// TIA Portal V19 export
FUNCTION "MFG OUTPUT SECTION" : Void   // FC10, LAD
{ S7_Optimized_Access := 'TRUE' }
// stored: SetENOAutomatically false
   VAR_TEMP   // added for the SCL form of the ladder/FBD networks
      _w1 : Bool;
   END_VAR
BEGIN

REGION Network 1: PSFV-1 – OPEN
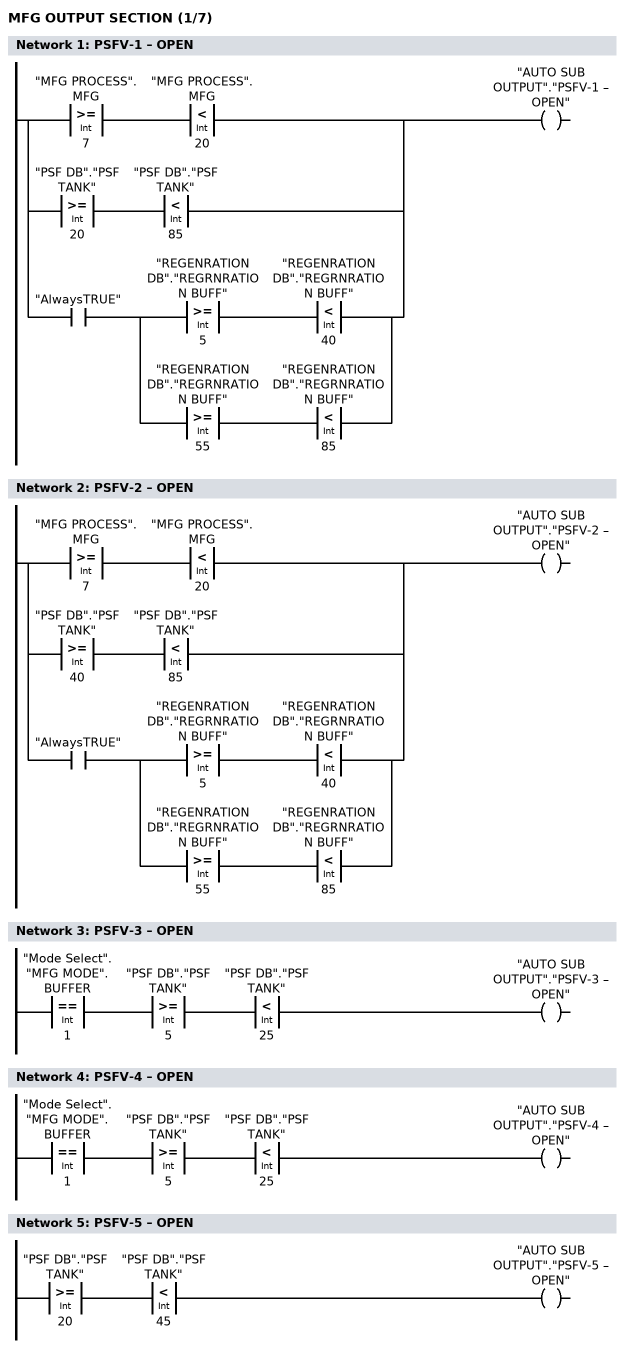
   RUNG wire#powerrail
      { S7_Templates := "SrcType := Int" } GE_Contact(in1 := "MFG PROCESS".MFG, in2 := 7)
      { S7_Templates := "SrcType := Int" } LT_Contact(in1 := "MFG PROCESS".MFG, in2 := 20)
      wire#w1
      Coil( "AUTO SUB OUTPUT"."PSFV-1 – OPEN" )
   END_RUNG
   RUNG wire#powerrail
      { S7_Templates := "SrcType := Int" } GE_Contact(in1 := "PSF DB"."PSF TANK", in2 := 20)
      { S7_Templates := "SrcType := Int" } LT_Contact(in1 := "PSF DB"."PSF TANK", in2 := 85)
   END_RUNG wire#w1
   RUNG wire#powerrail
      Contact( "AlwaysTRUE" )
      wire#w2
      { S7_Templates := "SrcType := Int" } GE_Contact(in1 := "REGENRATION DB"."REGRNRATION BUFF", in2 := 5)
      { S7_Templates := "SrcType := Int" } LT_Contact(in1 := "REGENRATION DB"."REGRNRATION BUFF", in2 := 40)
   END_RUNG wire#w1
   RUNG wire#w2
      { S7_Templates := "SrcType := Int" } GE_Contact(in1 := "REGENRATION DB"."REGRNRATION BUFF", in2 := 55)
      { S7_Templates := "SrcType := Int" } LT_Contact(in1 := "REGENRATION DB"."REGRNRATION BUFF", in2 := 85)
   END_RUNG wire#w1
   // the same network as SCL:
   "AUTO SUB OUTPUT"."PSFV-1 – OPEN" := (("MFG PROCESS".MFG >= 7) AND ("MFG PROCESS".MFG < 20)) OR (("PSF DB"."PSF TANK" >= 20) AND ("PSF DB"."PSF TANK" < 85)) OR ("AlwaysTRUE" AND ((("REGENRATION DB"."REGRNRATION BUFF" >= 5) AND ("REGENRATION DB"."REGRNRATION BUFF" < 40)) OR (("REGENRATION DB"."REGRNRATION BUFF" >= 55) AND ("REGENRATION DB"."REGRNRATION BUFF" < 85))));
END_REGION

REGION Network 2: PSFV-2 – OPEN
   RUNG wire#powerrail
      { S7_Templates := "SrcType := Int" } GE_Contact(in1 := "MFG PROCESS".MFG, in2 := 7)
      { S7_Templates := "SrcType := Int" } LT_Contact(in1 := "MFG PROCESS".MFG, in2 := 20)
      wire#w1
      Coil( "AUTO SUB OUTPUT"."PSFV-2 – OPEN" )
   END_RUNG
   RUNG wire#powerrail
      { S7_Templates := "SrcType := Int" } GE_Contact(in1 := "PSF DB"."PSF TANK", in2 := 40)
      { S7_Templates := "SrcType := Int" } LT_Contact(in1 := "PSF DB"."PSF TANK", in2 := 85)
   END_RUNG wire#w1
   RUNG wire#powerrail
      Contact( "AlwaysTRUE" )
      wire#w2
      { S7_Templates := "SrcType := Int" } GE_Contact(in1 := "REGENRATION DB"."REGRNRATION BUFF", in2 := 5)
      { S7_Templates := "SrcType := Int" } LT_Contact(in1 := "REGENRATION DB"."REGRNRATION BUFF", in2 := 40)
   END_RUNG wire#w1
   RUNG wire#w2
      { S7_Templates := "SrcType := Int" } GE_Contact(in1 := "REGENRATION DB"."REGRNRATION BUFF", in2 := 55)
      { S7_Templates := "SrcType := Int" } LT_Contact(in1 := "REGENRATION DB"."REGRNRATION BUFF", in2 := 85)
   END_RUNG wire#w1
   // the same network as SCL:
   "AUTO SUB OUTPUT"."PSFV-2 – OPEN" := (("MFG PROCESS".MFG >= 7) AND ("MFG PROCESS".MFG < 20)) OR (("PSF DB"."PSF TANK" >= 40) AND ("PSF DB"."PSF TANK" < 85)) OR ("AlwaysTRUE" AND ((("REGENRATION DB"."REGRNRATION BUFF" >= 5) AND ("REGENRATION DB"."REGRNRATION BUFF" < 40)) OR (("REGENRATION DB"."REGRNRATION BUFF" >= 55) AND ("REGENRATION DB"."REGRNRATION BUFF" < 85))));
END_REGION

REGION Network 3: PSFV-3 – OPEN
   RUNG wire#powerrail
      { S7_Templates := "SrcType := Int" } EQ_Contact(in1 := "Mode Select"."MFG MODE".BUFFER, in2 := 1)
      { S7_Templates := "SrcType := Int" } GE_Contact(in1 := "PSF DB"."PSF TANK", in2 := 5)
      { S7_Templates := "SrcType := Int" } LT_Contact(in1 := "PSF DB"."PSF TANK", in2 := 25)
      Coil( "AUTO SUB OUTPUT"."PSFV-3 – OPEN" )
   END_RUNG
   // the same network as SCL:
   "AUTO SUB OUTPUT"."PSFV-3 – OPEN" := ("Mode Select"."MFG MODE".BUFFER = 1) AND ("PSF DB"."PSF TANK" >= 5) AND ("PSF DB"."PSF TANK" < 25);
END_REGION

REGION Network 4: PSFV-4 – OPEN
   RUNG wire#powerrail
      { S7_Templates := "SrcType := Int" } EQ_Contact(in1 := "Mode Select"."MFG MODE".BUFFER, in2 := 1)
      { S7_Templates := "SrcType := Int" } GE_Contact(in1 := "PSF DB"."PSF TANK", in2 := 5)
      { S7_Templates := "SrcType := Int" } LT_Contact(in1 := "PSF DB"."PSF TANK", in2 := 25)
      Coil( "AUTO SUB OUTPUT"."PSFV-4 – OPEN" )
   END_RUNG
   // the same network as SCL:
   "AUTO SUB OUTPUT"."PSFV-4 – OPEN" := ("Mode Select"."MFG MODE".BUFFER = 1) AND ("PSF DB"."PSF TANK" >= 5) AND ("PSF DB"."PSF TANK" < 25);
END_REGION

REGION Network 5: PSFV-5 – OPEN
   RUNG wire#powerrail
      { S7_Templates := "SrcType := Int" } GE_Contact(in1 := "PSF DB"."PSF TANK", in2 := 20)
      { S7_Templates := "SrcType := Int" } LT_Contact(in1 := "PSF DB"."PSF TANK", in2 := 45)
      Coil( "AUTO SUB OUTPUT"."PSFV-5 – OPEN" )
   END_RUNG
   // the same network as SCL:
   "AUTO SUB OUTPUT"."PSFV-5 – OPEN" := ("PSF DB"."PSF TANK" >= 20) AND ("PSF DB"."PSF TANK" < 45);
END_REGION

REGION Network 6: PSFV-6 – OPEN
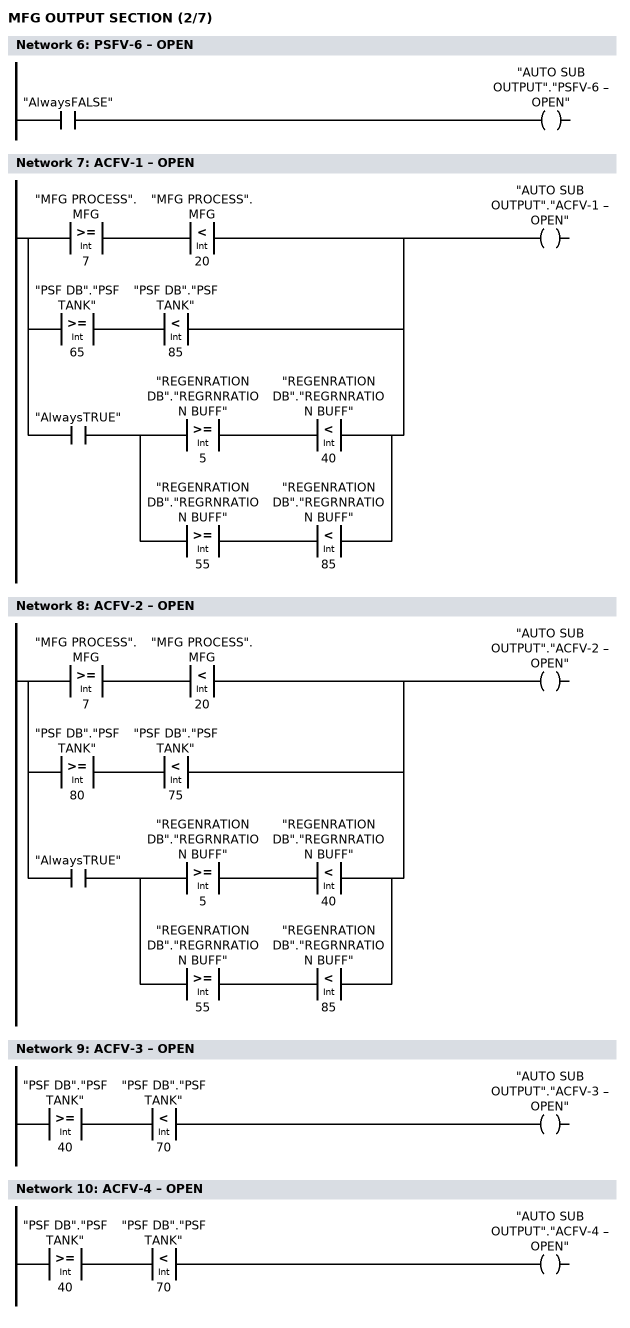
   RUNG wire#powerrail
      Contact( "AlwaysFALSE" )
      Coil( "AUTO SUB OUTPUT"."PSFV-6 – OPEN" )
   END_RUNG
   // the same network as SCL:
   "AUTO SUB OUTPUT"."PSFV-6 – OPEN" := "AlwaysFALSE";
END_REGION

REGION Network 7: ACFV-1 – OPEN
   RUNG wire#powerrail
      { S7_Templates := "SrcType := Int" } GE_Contact(in1 := "MFG PROCESS".MFG, in2 := 7)
      { S7_Templates := "SrcType := Int" } LT_Contact(in1 := "MFG PROCESS".MFG, in2 := 20)
      wire#w1
      Coil( "AUTO SUB OUTPUT"."ACFV-1 – OPEN" )
   END_RUNG
   RUNG wire#powerrail
      { S7_Templates := "SrcType := Int" } GE_Contact(in1 := "PSF DB"."PSF TANK", in2 := 65)
      { S7_Templates := "SrcType := Int" } LT_Contact(in1 := "PSF DB"."PSF TANK", in2 := 85)
   END_RUNG wire#w1
   RUNG wire#powerrail
      Contact( "AlwaysTRUE" )
      wire#w2
      { S7_Templates := "SrcType := Int" } GE_Contact(in1 := "REGENRATION DB"."REGRNRATION BUFF", in2 := 5)
      { S7_Templates := "SrcType := Int" } LT_Contact(in1 := "REGENRATION DB"."REGRNRATION BUFF", in2 := 40)
   END_RUNG wire#w1
   RUNG wire#w2
      { S7_Templates := "SrcType := Int" } GE_Contact(in1 := "REGENRATION DB"."REGRNRATION BUFF", in2 := 55)
      { S7_Templates := "SrcType := Int" } LT_Contact(in1 := "REGENRATION DB"."REGRNRATION BUFF", in2 := 85)
   END_RUNG wire#w1
   // the same network as SCL:
   "AUTO SUB OUTPUT"."ACFV-1 – OPEN" := (("MFG PROCESS".MFG >= 7) AND ("MFG PROCESS".MFG < 20)) OR (("PSF DB"."PSF TANK" >= 65) AND ("PSF DB"."PSF TANK" < 85)) OR ("AlwaysTRUE" AND ((("REGENRATION DB"."REGRNRATION BUFF" >= 5) AND ("REGENRATION DB"."REGRNRATION BUFF" < 40)) OR (("REGENRATION DB"."REGRNRATION BUFF" >= 55) AND ("REGENRATION DB"."REGRNRATION BUFF" < 85))));
END_REGION

REGION Network 8: ACFV-2 – OPEN
   RUNG wire#powerrail
      { S7_Templates := "SrcType := Int" } GE_Contact(in1 := "MFG PROCESS".MFG, in2 := 7)
      { S7_Templates := "SrcType := Int" } LT_Contact(in1 := "MFG PROCESS".MFG, in2 := 20)
      wire#w1
      Coil( "AUTO SUB OUTPUT"."ACFV-2 – OPEN" )
   END_RUNG
   RUNG wire#powerrail
      { S7_Templates := "SrcType := Int" } GE_Contact(in1 := "PSF DB"."PSF TANK", in2 := 80)
      { S7_Templates := "SrcType := Int" } LT_Contact(in1 := "PSF DB"."PSF TANK", in2 := 75)
   END_RUNG wire#w1
   RUNG wire#powerrail
      Contact( "AlwaysTRUE" )
      wire#w2
      { S7_Templates := "SrcType := Int" } GE_Contact(in1 := "REGENRATION DB"."REGRNRATION BUFF", in2 := 5)
      { S7_Templates := "SrcType := Int" } LT_Contact(in1 := "REGENRATION DB"."REGRNRATION BUFF", in2 := 40)
   END_RUNG wire#w1
   RUNG wire#w2
      { S7_Templates := "SrcType := Int" } GE_Contact(in1 := "REGENRATION DB"."REGRNRATION BUFF", in2 := 55)
      { S7_Templates := "SrcType := Int" } LT_Contact(in1 := "REGENRATION DB"."REGRNRATION BUFF", in2 := 85)
   END_RUNG wire#w1
   // the same network as SCL:
   "AUTO SUB OUTPUT"."ACFV-2 – OPEN" := (("MFG PROCESS".MFG >= 7) AND ("MFG PROCESS".MFG < 20)) OR (("PSF DB"."PSF TANK" >= 80) AND ("PSF DB"."PSF TANK" < 75)) OR ("AlwaysTRUE" AND ((("REGENRATION DB"."REGRNRATION BUFF" >= 5) AND ("REGENRATION DB"."REGRNRATION BUFF" < 40)) OR (("REGENRATION DB"."REGRNRATION BUFF" >= 55) AND ("REGENRATION DB"."REGRNRATION BUFF" < 85))));
END_REGION

REGION Network 9: ACFV-3 – OPEN
   RUNG wire#powerrail
      { S7_Templates := "SrcType := Int" } GE_Contact(in1 := "PSF DB"."PSF TANK", in2 := 40)
      { S7_Templates := "SrcType := Int" } LT_Contact(in1 := "PSF DB"."PSF TANK", in2 := 70)
      Coil( "AUTO SUB OUTPUT"."ACFV-3 – OPEN" )
   END_RUNG
   // the same network as SCL:
   "AUTO SUB OUTPUT"."ACFV-3 – OPEN" := ("PSF DB"."PSF TANK" >= 40) AND ("PSF DB"."PSF TANK" < 70);
END_REGION

REGION Network 10: ACFV-4 – OPEN
   RUNG wire#powerrail
      { S7_Templates := "SrcType := Int" } GE_Contact(in1 := "PSF DB"."PSF TANK", in2 := 40)
      { S7_Templates := "SrcType := Int" } LT_Contact(in1 := "PSF DB"."PSF TANK", in2 := 70)
      Coil( "AUTO SUB OUTPUT"."ACFV-4 – OPEN" )
   END_RUNG
   // the same network as SCL:
   "AUTO SUB OUTPUT"."ACFV-4 – OPEN" := ("PSF DB"."PSF TANK" >= 40) AND ("PSF DB"."PSF TANK" < 70);
END_REGION

REGION Network 11: ACFV-5 – OPEN
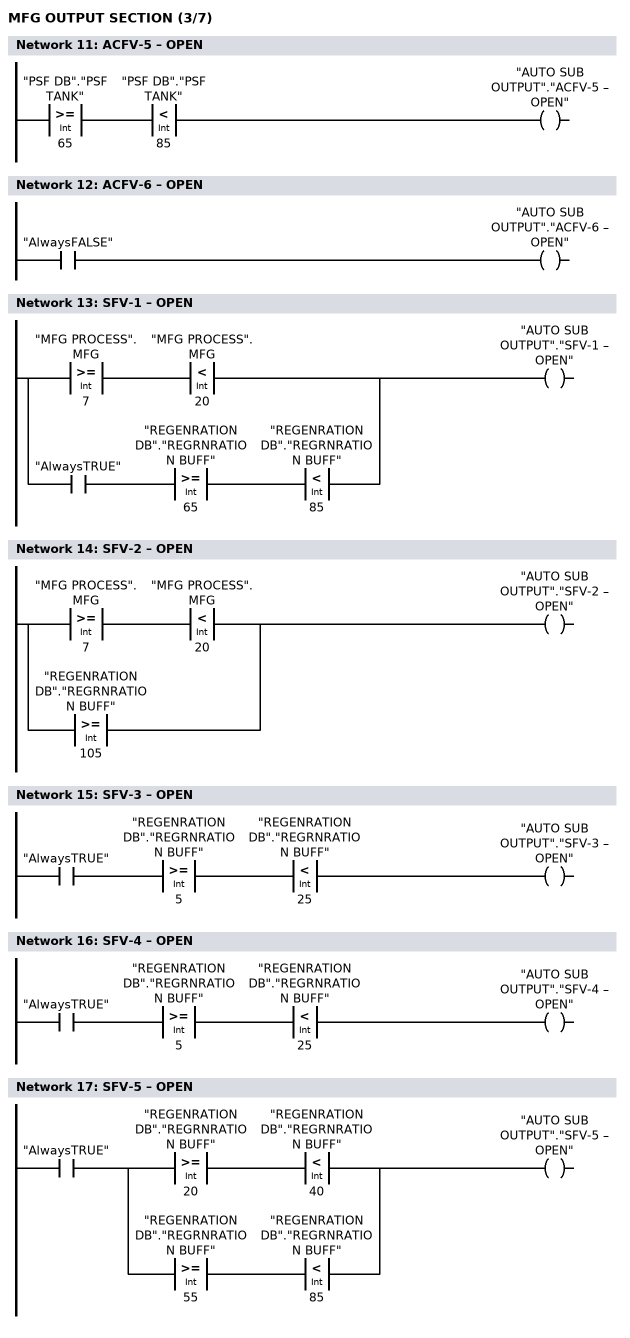
   RUNG wire#powerrail
      { S7_Templates := "SrcType := Int" } GE_Contact(in1 := "PSF DB"."PSF TANK", in2 := 65)
      { S7_Templates := "SrcType := Int" } LT_Contact(in1 := "PSF DB"."PSF TANK", in2 := 85)
      Coil( "AUTO SUB OUTPUT"."ACFV-5 – OPEN" )
   END_RUNG
   // the same network as SCL:
   "AUTO SUB OUTPUT"."ACFV-5 – OPEN" := ("PSF DB"."PSF TANK" >= 65) AND ("PSF DB"."PSF TANK" < 85);
END_REGION

REGION Network 12: ACFV-6 – OPEN
   RUNG wire#powerrail
      Contact( "AlwaysFALSE" )
      Coil( "AUTO SUB OUTPUT"."ACFV-6 – OPEN" )
   END_RUNG
   // the same network as SCL:
   "AUTO SUB OUTPUT"."ACFV-6 – OPEN" := "AlwaysFALSE";
END_REGION

REGION Network 13: SFV-1 – OPEN
   RUNG wire#powerrail
      { S7_Templates := "SrcType := Int" } GE_Contact(in1 := "MFG PROCESS".MFG, in2 := 7)
      { S7_Templates := "SrcType := Int" } LT_Contact(in1 := "MFG PROCESS".MFG, in2 := 20)
      wire#w1
      Coil( "AUTO SUB OUTPUT"."SFV-1 – OPEN" )
   END_RUNG
   RUNG wire#powerrail
      Contact( "AlwaysTRUE" )
      { S7_Templates := "SrcType := Int" } GE_Contact(in1 := "REGENRATION DB"."REGRNRATION BUFF", in2 := 65)
      { S7_Templates := "SrcType := Int" } LT_Contact(in1 := "REGENRATION DB"."REGRNRATION BUFF", in2 := 85)
   END_RUNG wire#w1
   // the same network as SCL:
   "AUTO SUB OUTPUT"."SFV-1 – OPEN" := (("MFG PROCESS".MFG >= 7) AND ("MFG PROCESS".MFG < 20)) OR ("AlwaysTRUE" AND ("REGENRATION DB"."REGRNRATION BUFF" >= 65) AND ("REGENRATION DB"."REGRNRATION BUFF" < 85));
END_REGION

REGION Network 14: SFV-2 – OPEN
   RUNG wire#powerrail
      { S7_Templates := "SrcType := Int" } GE_Contact(in1 := "MFG PROCESS".MFG, in2 := 7)
      { S7_Templates := "SrcType := Int" } LT_Contact(in1 := "MFG PROCESS".MFG, in2 := 20)
      wire#w1
      Coil( "AUTO SUB OUTPUT"."SFV-2 – OPEN" )
   END_RUNG
   RUNG wire#powerrail
      { S7_Templates := "SrcType := Int" } GE_Contact(in1 := "REGENRATION DB"."REGRNRATION BUFF", in2 := 105)
   END_RUNG wire#w1
   // the same network as SCL:
   "AUTO SUB OUTPUT"."SFV-2 – OPEN" := (("MFG PROCESS".MFG >= 7) AND ("MFG PROCESS".MFG < 20)) OR ("REGENRATION DB"."REGRNRATION BUFF" >= 105);
END_REGION

REGION Network 15: SFV-3 – OPEN
   RUNG wire#powerrail
      Contact( "AlwaysTRUE" )
      { S7_Templates := "SrcType := Int" } GE_Contact(in1 := "REGENRATION DB"."REGRNRATION BUFF", in2 := 5)
      { S7_Templates := "SrcType := Int" } LT_Contact(in1 := "REGENRATION DB"."REGRNRATION BUFF", in2 := 25)
      Coil( "AUTO SUB OUTPUT"."SFV-3 – OPEN" )
   END_RUNG
   // the same network as SCL:
   "AUTO SUB OUTPUT"."SFV-3 – OPEN" := "AlwaysTRUE" AND ("REGENRATION DB"."REGRNRATION BUFF" >= 5) AND ("REGENRATION DB"."REGRNRATION BUFF" < 25);
END_REGION

REGION Network 16: SFV-4 – OPEN
   RUNG wire#powerrail
      Contact( "AlwaysTRUE" )
      { S7_Templates := "SrcType := Int" } GE_Contact(in1 := "REGENRATION DB"."REGRNRATION BUFF", in2 := 5)
      { S7_Templates := "SrcType := Int" } LT_Contact(in1 := "REGENRATION DB"."REGRNRATION BUFF", in2 := 25)
      Coil( "AUTO SUB OUTPUT"."SFV-4 – OPEN" )
   END_RUNG
   // the same network as SCL:
   "AUTO SUB OUTPUT"."SFV-4 – OPEN" := "AlwaysTRUE" AND ("REGENRATION DB"."REGRNRATION BUFF" >= 5) AND ("REGENRATION DB"."REGRNRATION BUFF" < 25);
END_REGION

REGION Network 17: SFV-5 – OPEN
   RUNG wire#powerrail
      Contact( "AlwaysTRUE" )
      wire#w1
      { S7_Templates := "SrcType := Int" } GE_Contact(in1 := "REGENRATION DB"."REGRNRATION BUFF", in2 := 20)
      { S7_Templates := "SrcType := Int" } LT_Contact(in1 := "REGENRATION DB"."REGRNRATION BUFF", in2 := 40)
      wire#w2
      Coil( "AUTO SUB OUTPUT"."SFV-5 – OPEN" )
   END_RUNG
   RUNG wire#w1
      { S7_Templates := "SrcType := Int" } GE_Contact(in1 := "REGENRATION DB"."REGRNRATION BUFF", in2 := 55)
      { S7_Templates := "SrcType := Int" } LT_Contact(in1 := "REGENRATION DB"."REGRNRATION BUFF", in2 := 85)
   END_RUNG wire#w2
   // the same network as SCL:
   "AUTO SUB OUTPUT"."SFV-5 – OPEN" := "AlwaysTRUE" AND ((("REGENRATION DB"."REGRNRATION BUFF" >= 20) AND ("REGENRATION DB"."REGRNRATION BUFF" < 40)) OR (("REGENRATION DB"."REGRNRATION BUFF" >= 55) AND ("REGENRATION DB"."REGRNRATION BUFF" < 85)));
END_REGION

REGION Network 18: SFV-6 – OPEN
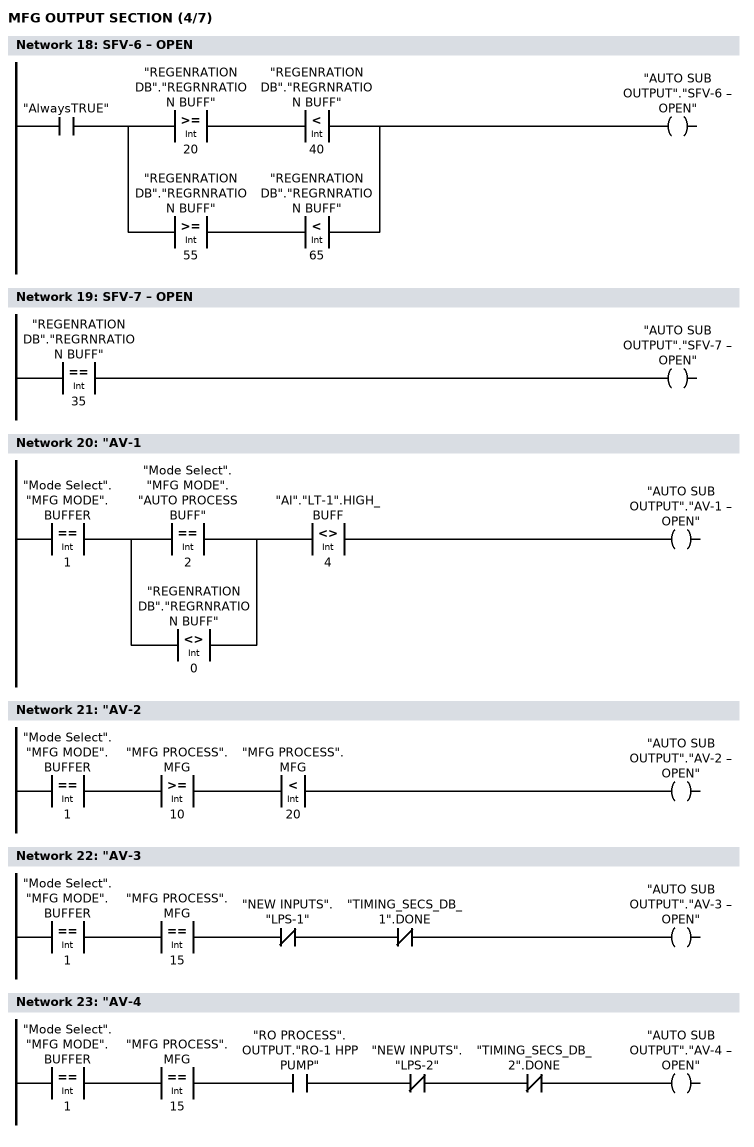
   RUNG wire#powerrail
      Contact( "AlwaysTRUE" )
      wire#w1
      { S7_Templates := "SrcType := Int" } GE_Contact(in1 := "REGENRATION DB"."REGRNRATION BUFF", in2 := 20)
      { S7_Templates := "SrcType := Int" } LT_Contact(in1 := "REGENRATION DB"."REGRNRATION BUFF", in2 := 40)
      wire#w2
      Coil( "AUTO SUB OUTPUT"."SFV-6 – OPEN" )
   END_RUNG
   RUNG wire#w1
      { S7_Templates := "SrcType := Int" } GE_Contact(in1 := "REGENRATION DB"."REGRNRATION BUFF", in2 := 55)
      { S7_Templates := "SrcType := Int" } LT_Contact(in1 := "REGENRATION DB"."REGRNRATION BUFF", in2 := 65)
   END_RUNG wire#w2
   // the same network as SCL:
   "AUTO SUB OUTPUT"."SFV-6 – OPEN" := "AlwaysTRUE" AND ((("REGENRATION DB"."REGRNRATION BUFF" >= 20) AND ("REGENRATION DB"."REGRNRATION BUFF" < 40)) OR (("REGENRATION DB"."REGRNRATION BUFF" >= 55) AND ("REGENRATION DB"."REGRNRATION BUFF" < 65)));
END_REGION

REGION Network 19: SFV-7 – OPEN
   RUNG wire#powerrail
      { S7_Templates := "SrcType := Int" } EQ_Contact(in1 := "REGENRATION DB"."REGRNRATION BUFF", in2 := 35)
      Coil( "AUTO SUB OUTPUT"."SFV-7 – OPEN" )
   END_RUNG
   // the same network as SCL:
   "AUTO SUB OUTPUT"."SFV-7 – OPEN" := "REGENRATION DB"."REGRNRATION BUFF" = 35;
END_REGION

REGION Network 20: "AV-1
   RUNG wire#powerrail
      { S7_Templates := "SrcType := Int" } EQ_Contact(in1 := "Mode Select"."MFG MODE".BUFFER, in2 := 1)
      wire#w1
      { S7_Templates := "SrcType := Int" } EQ_Contact(in1 := "Mode Select"."MFG MODE"."AUTO PROCESS BUFF", in2 := 2)
      wire#w2
      { S7_Templates := "SrcType := Int" } NE_Contact(in1 := "AI"."LT-1".HIGH_BUFF, in2 := 4)
      Coil( "AUTO SUB OUTPUT"."AV-1 – OPEN" )
   END_RUNG
   RUNG wire#w1
      { S7_Templates := "SrcType := Int" } NE_Contact(in1 := "REGENRATION DB"."REGRNRATION BUFF", in2 := 0)
   END_RUNG wire#w2
   // the same network as SCL:
   "AUTO SUB OUTPUT"."AV-1 – OPEN" := ("Mode Select"."MFG MODE".BUFFER = 1) AND (("Mode Select"."MFG MODE"."AUTO PROCESS BUFF" = 2) OR ("REGENRATION DB"."REGRNRATION BUFF" <> 0)) AND ("AI"."LT-1".HIGH_BUFF <> 4);
END_REGION

REGION Network 21: "AV-2
   RUNG wire#powerrail
      { S7_Templates := "SrcType := Int" } EQ_Contact(in1 := "Mode Select"."MFG MODE".BUFFER, in2 := 1)
      { S7_Templates := "SrcType := Int" } GE_Contact(in1 := "MFG PROCESS".MFG, in2 := 10)
      { S7_Templates := "SrcType := Int" } LT_Contact(in1 := "MFG PROCESS".MFG, in2 := 20)
      Coil( "AUTO SUB OUTPUT"."AV-2 – OPEN" )
   END_RUNG
   // the same network as SCL:
   "AUTO SUB OUTPUT"."AV-2 – OPEN" := ("Mode Select"."MFG MODE".BUFFER = 1) AND ("MFG PROCESS".MFG >= 10) AND ("MFG PROCESS".MFG < 20);
END_REGION

REGION Network 22: "AV-3
   RUNG wire#powerrail
      { S7_Templates := "SrcType := Int" } EQ_Contact(in1 := "Mode Select"."MFG MODE".BUFFER, in2 := 1)
      { S7_Templates := "SrcType := Int" } EQ_Contact(in1 := "MFG PROCESS".MFG, in2 := 15)
      I_Contact( "NEW INPUTS"."LPS-1" )
      I_Contact( "TIMING_SECS_DB_1".DONE )
      Coil( "AUTO SUB OUTPUT"."AV-3 – OPEN" )
   END_RUNG
   // the same network as SCL:
   "AUTO SUB OUTPUT"."AV-3 – OPEN" := ("Mode Select"."MFG MODE".BUFFER = 1) AND ("MFG PROCESS".MFG = 15) AND NOT "NEW INPUTS"."LPS-1" AND NOT "TIMING_SECS_DB_1".DONE;
END_REGION

REGION Network 23: "AV-4
   RUNG wire#powerrail
      { S7_Templates := "SrcType := Int" } EQ_Contact(in1 := "Mode Select"."MFG MODE".BUFFER, in2 := 1)
      { S7_Templates := "SrcType := Int" } EQ_Contact(in1 := "MFG PROCESS".MFG, in2 := 15)
      Contact( "RO PROCESS".OUTPUT."RO-1 HPP PUMP" )
      I_Contact( "NEW INPUTS"."LPS-2" )
      I_Contact( "TIMING_SECS_DB_2".DONE )
      Coil( "AUTO SUB OUTPUT"."AV-4 – OPEN" )
   END_RUNG
   // the same network as SCL:
   "AUTO SUB OUTPUT"."AV-4 – OPEN" := ("Mode Select"."MFG MODE".BUFFER = 1) AND ("MFG PROCESS".MFG = 15) AND "RO PROCESS".OUTPUT."RO-1 HPP PUMP" AND NOT "NEW INPUTS"."LPS-2" AND NOT "TIMING_SECS_DB_2".DONE;
END_REGION

REGION Network 24: DP-1
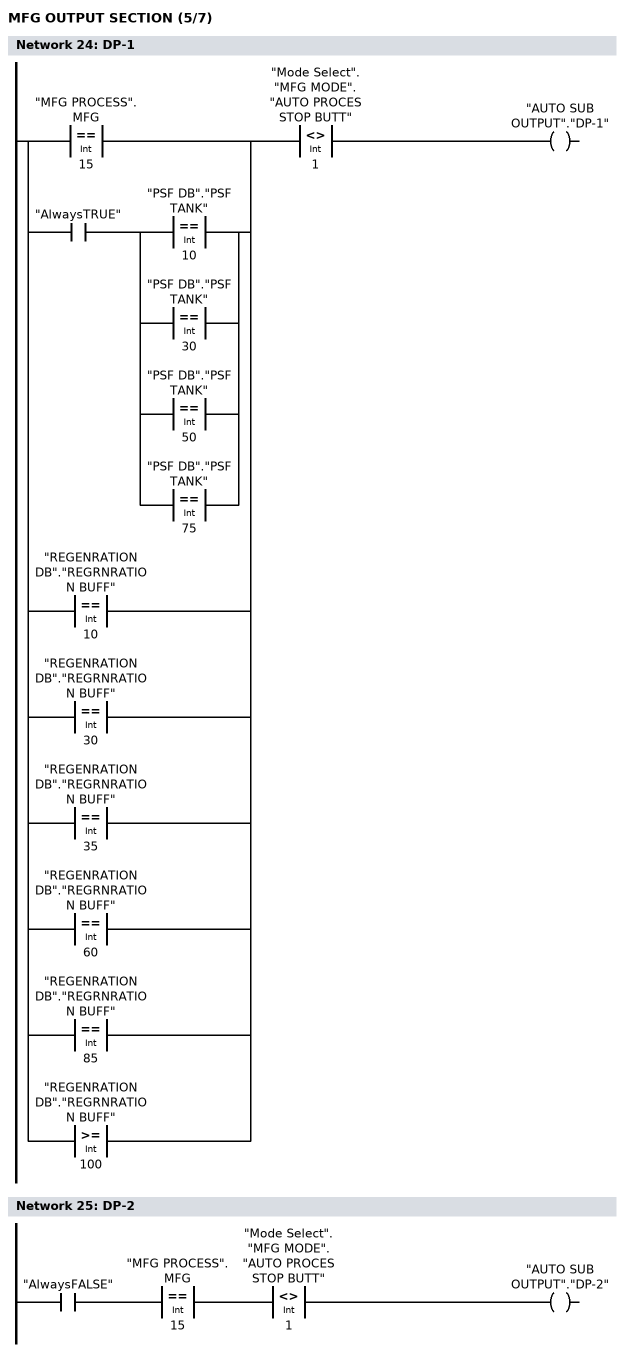
   RUNG wire#powerrail
      { S7_Templates := "SrcType := Int" } EQ_Contact(in1 := "MFG PROCESS".MFG, in2 := 15)
      wire#w1
      { S7_Templates := "SrcType := Int" } NE_Contact(in1 := "Mode Select"."MFG MODE"."AUTO PROCES STOP BUTT", in2 := 1)
      Coil( "AUTO SUB OUTPUT"."DP-1" )
   END_RUNG
   RUNG wire#powerrail
      Contact( "AlwaysTRUE" )
      wire#w2
      { S7_Templates := "SrcType := Int" } EQ_Contact(in1 := "PSF DB"."PSF TANK", in2 := 10)
   END_RUNG wire#w1
   RUNG wire#w2
      { S7_Templates := "SrcType := Int" } EQ_Contact(in1 := "PSF DB"."PSF TANK", in2 := 30)
   END_RUNG wire#w1
   RUNG wire#w2
      { S7_Templates := "SrcType := Int" } EQ_Contact(in1 := "PSF DB"."PSF TANK", in2 := 50)
   END_RUNG wire#w1
   RUNG wire#w2
      { S7_Templates := "SrcType := Int" } EQ_Contact(in1 := "PSF DB"."PSF TANK", in2 := 75)
   END_RUNG wire#w1
   RUNG wire#powerrail
      { S7_Templates := "SrcType := Int" } EQ_Contact(in1 := "REGENRATION DB"."REGRNRATION BUFF", in2 := 10)
   END_RUNG wire#w1
   RUNG wire#powerrail
      { S7_Templates := "SrcType := Int" } EQ_Contact(in1 := "REGENRATION DB"."REGRNRATION BUFF", in2 := 30)
   END_RUNG wire#w1
   RUNG wire#powerrail
      { S7_Templates := "SrcType := Int" } EQ_Contact(in1 := "REGENRATION DB"."REGRNRATION BUFF", in2 := 35)
   END_RUNG wire#w1
   RUNG wire#powerrail
      { S7_Templates := "SrcType := Int" } EQ_Contact(in1 := "REGENRATION DB"."REGRNRATION BUFF", in2 := 60)
   END_RUNG wire#w1
   RUNG wire#powerrail
      { S7_Templates := "SrcType := Int" } EQ_Contact(in1 := "REGENRATION DB"."REGRNRATION BUFF", in2 := 85)
   END_RUNG wire#w1
   RUNG wire#powerrail
      { S7_Templates := "SrcType := Int" } GE_Contact(in1 := "REGENRATION DB"."REGRNRATION BUFF", in2 := 100)
   END_RUNG wire#w1
   // the same network as SCL:
   "AUTO SUB OUTPUT"."DP-1" := (("MFG PROCESS".MFG = 15) OR ("AlwaysTRUE" AND (("PSF DB"."PSF TANK" = 10) OR ("PSF DB"."PSF TANK" = 30) OR ("PSF DB"."PSF TANK" = 50) OR ("PSF DB"."PSF TANK" = 75))) OR ("REGENRATION DB"."REGRNRATION BUFF" = 10) OR ("REGENRATION DB"."REGRNRATION BUFF" = 30) OR ("REGENRATION DB"."REGRNRATION BUFF" = 35) OR ("REGENRATION DB"."REGRNRATION BUFF" = 60) OR ("REGENRATION DB"."REGRNRATION BUFF" = 85) OR ("REGENRATION DB"."REGRNRATION BUFF" >= 100)) AND ("Mode Select"."MFG MODE"."AUTO PROCES STOP BUTT" <> 1);
END_REGION

REGION Network 25: DP-2
   RUNG wire#powerrail
      Contact( "AlwaysFALSE" )
      { S7_Templates := "SrcType := Int" } EQ_Contact(in1 := "MFG PROCESS".MFG, in2 := 15)
      { S7_Templates := "SrcType := Int" } NE_Contact(in1 := "Mode Select"."MFG MODE"."AUTO PROCES STOP BUTT", in2 := 1)
      Coil( "AUTO SUB OUTPUT"."DP-2" )
   END_RUNG
   // the same network as SCL:
   "AUTO SUB OUTPUT"."DP-2" := "AlwaysFALSE" AND ("MFG PROCESS".MFG = 15) AND ("Mode Select"."MFG MODE"."AUTO PROCES STOP BUTT" <> 1);
END_REGION

REGION Network 26: DP-3
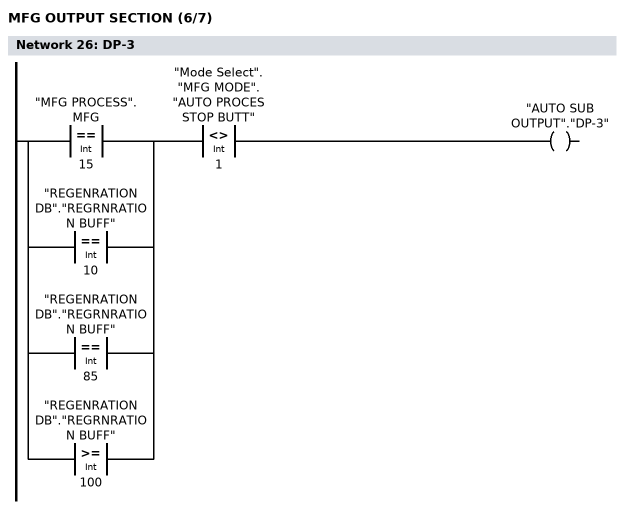
   RUNG wire#powerrail
      { S7_Templates := "SrcType := Int" } EQ_Contact(in1 := "MFG PROCESS".MFG, in2 := 15)
      wire#w1
      { S7_Templates := "SrcType := Int" } NE_Contact(in1 := "Mode Select"."MFG MODE"."AUTO PROCES STOP BUTT", in2 := 1)
      Coil( "AUTO SUB OUTPUT"."DP-3" )
   END_RUNG
   RUNG wire#powerrail
      { S7_Templates := "SrcType := Int" } EQ_Contact(in1 := "REGENRATION DB"."REGRNRATION BUFF", in2 := 10)
   END_RUNG wire#w1
   RUNG wire#powerrail
      { S7_Templates := "SrcType := Int" } EQ_Contact(in1 := "REGENRATION DB"."REGRNRATION BUFF", in2 := 85)
   END_RUNG wire#w1
   RUNG wire#powerrail
      { S7_Templates := "SrcType := Int" } GE_Contact(in1 := "REGENRATION DB"."REGRNRATION BUFF", in2 := 100)
   END_RUNG wire#w1
   // the same network as SCL:
   "AUTO SUB OUTPUT"."DP-3" := (("MFG PROCESS".MFG = 15) OR ("REGENRATION DB"."REGRNRATION BUFF" = 10) OR ("REGENRATION DB"."REGRNRATION BUFF" = 85) OR ("REGENRATION DB"."REGRNRATION BUFF" >= 100)) AND ("Mode Select"."MFG MODE"."AUTO PROCES STOP BUTT" <> 1);
END_REGION

REGION Network 27: FEED PUMP
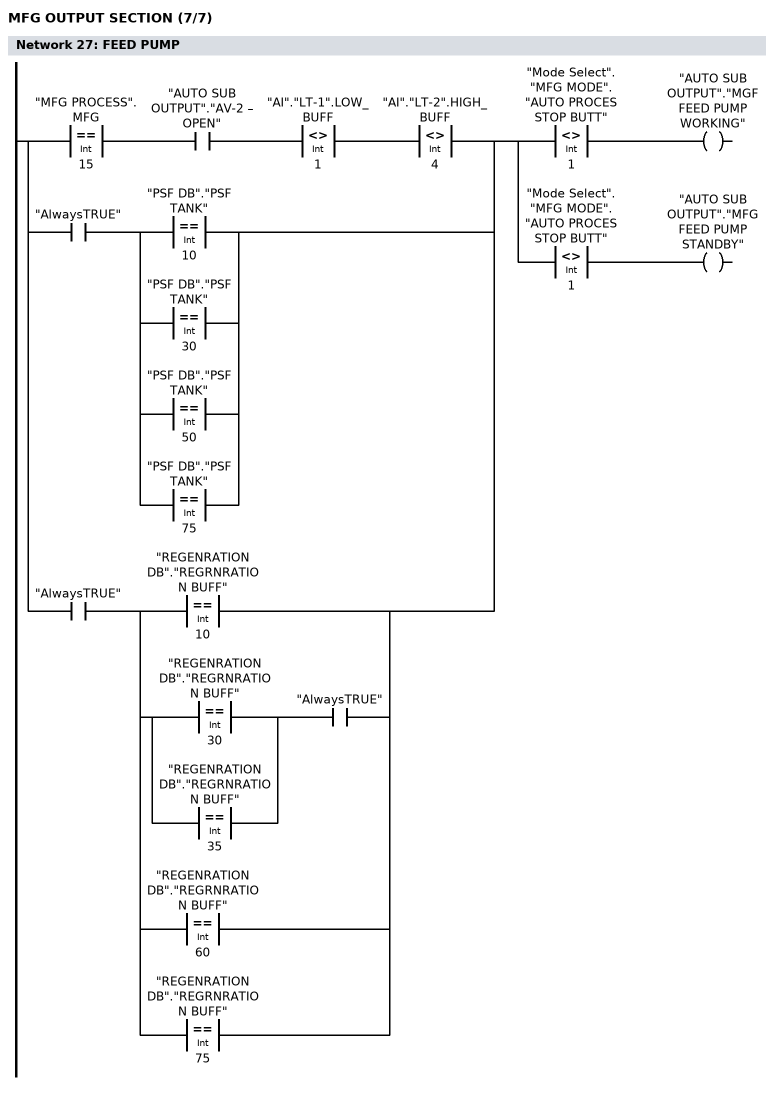
   RUNG wire#powerrail
      { S7_Templates := "SrcType := Int" } EQ_Contact(in1 := "MFG PROCESS".MFG, in2 := 15)
      Contact( "AUTO SUB OUTPUT"."AV-2 – OPEN" )
      { S7_Templates := "SrcType := Int" } NE_Contact(in1 := "AI"."LT-1".LOW_BUFF, in2 := 1)
      { S7_Templates := "SrcType := Int" } NE_Contact(in1 := "AI"."LT-2".HIGH_BUFF, in2 := 4)
      wire#w1
      { S7_Templates := "SrcType := Int" } NE_Contact(in1 := "Mode Select"."MFG MODE"."AUTO PROCES STOP BUTT", in2 := 1)
      Coil( "AUTO SUB OUTPUT"."MGF FEED PUMP WORKING" )
   END_RUNG
   RUNG wire#powerrail
      Contact( "AlwaysTRUE" )
      wire#w2
      { S7_Templates := "SrcType := Int" } EQ_Contact(in1 := "PSF DB"."PSF TANK", in2 := 10)
   END_RUNG wire#w1
   RUNG wire#w2
      { S7_Templates := "SrcType := Int" } EQ_Contact(in1 := "PSF DB"."PSF TANK", in2 := 30)
   END_RUNG wire#w1
   RUNG wire#w2
      { S7_Templates := "SrcType := Int" } EQ_Contact(in1 := "PSF DB"."PSF TANK", in2 := 50)
   END_RUNG wire#w1
   RUNG wire#w2
      { S7_Templates := "SrcType := Int" } EQ_Contact(in1 := "PSF DB"."PSF TANK", in2 := 75)
   END_RUNG wire#w1
   RUNG wire#powerrail
      Contact( "AlwaysTRUE" )
      wire#w3
      { S7_Templates := "SrcType := Int" } EQ_Contact(in1 := "REGENRATION DB"."REGRNRATION BUFF", in2 := 10)
   END_RUNG wire#w1
   RUNG wire#w3
      { S7_Templates := "SrcType := Int" } EQ_Contact(in1 := "REGENRATION DB"."REGRNRATION BUFF", in2 := 30)
      wire#w4
      Contact( "AlwaysTRUE" )
   END_RUNG wire#w1
   RUNG wire#w3
      { S7_Templates := "SrcType := Int" } EQ_Contact(in1 := "REGENRATION DB"."REGRNRATION BUFF", in2 := 35)
   END_RUNG wire#w4
   RUNG wire#w3
      { S7_Templates := "SrcType := Int" } EQ_Contact(in1 := "REGENRATION DB"."REGRNRATION BUFF", in2 := 60)
   END_RUNG wire#w1
   RUNG wire#w3
      { S7_Templates := "SrcType := Int" } EQ_Contact(in1 := "REGENRATION DB"."REGRNRATION BUFF", in2 := 75)
   END_RUNG wire#w1
   RUNG wire#w1
      { S7_Templates := "SrcType := Int" } NE_Contact(in1 := "Mode Select"."MFG MODE"."AUTO PROCES STOP BUTT", in2 := 1)
      Coil( "AUTO SUB OUTPUT"."MFG FEED PUMP STANDBY" )
   END_RUNG
   // the same network as SCL:
   #_w1 := (("MFG PROCESS".MFG = 15) AND "AUTO SUB OUTPUT"."AV-2 – OPEN" AND ("AI"."LT-1".LOW_BUFF <> 1) AND ("AI"."LT-2".HIGH_BUFF <> 4)) OR ("AlwaysTRUE" AND (("PSF DB"."PSF TANK" = 10) OR ("PSF DB"."PSF TANK" = 30) OR ("PSF DB"."PSF TANK" = 50) OR ("PSF DB"."PSF TANK" = 75))) OR ("AlwaysTRUE" AND (("REGENRATION DB"."REGRNRATION BUFF" = 10) OR ((("REGENRATION DB"."REGRNRATION BUFF" = 30) OR ("REGENRATION DB"."REGRNRATION BUFF" = 35)) AND "AlwaysTRUE") OR ("REGENRATION DB"."REGRNRATION BUFF" = 60) OR ("REGENRATION DB"."REGRNRATION BUFF" = 75)));
   "AUTO SUB OUTPUT"."MGF FEED PUMP WORKING" := #_w1 AND ("Mode Select"."MFG MODE"."AUTO PROCES STOP BUTT" <> 1);
   "AUTO SUB OUTPUT"."MFG FEED PUMP STANDBY" := #_w1 AND ("Mode Select"."MFG MODE"."AUTO PROCES STOP BUTT" <> 1);
END_REGION
END_FUNCTION
